{attribute 'qualified_only'}
{attribute 'strict'}
{attribute 'to_string'}
TYPE LinearStates :
(
	Initialising,
	Start_Homing,
	Homing,
	Idle,
	Start_Move,
	Moving,
	Error
);
END_TYPE

(* stored: Version 1.1.0.1, ProductVersion 3.1.4024.12
   DUT LinearStates: Id {92b77659-70d9-4b3c-bd1f-796ed907fd91} *)
